TYPE UDT_Fault :
STRUCT
	Active 			: BOOL := FALSE;
	FaultType 		: E_FaultTypes;
	Description 	: STRING;
END_STRUCT
END_TYPE

(* stored: Version 1.1.0.1, ProductVersion 3.1.4024.11
   DUT UDT_Fault: Id {4279845d-19ed-4754-876f-7c5a27f78cb3} *)
